INTERFACE I_DS402Common EXTENDS __SYSTEM.IQueryInterface, I_Output, I_Home

METHOD OperationMode
VAR_INPUT
END_VAR
END_METHOD

END_INTERFACE

(* stored: Version 1.1.0.1
   Itf I_DS402Common: Id {aa475227-9d3f-411c-89b0-156fd641ec44}
   Method OperationMode: Id {504f5dfc-7c72-43e8-a5ad-0a8e8e7ecf41} *)
